FUNCTION_BLOCK FB_AnalogInput
(*
    Converts the integer from an analog input terminal to a real unit value (e.g., volts)
    2019-10-09 Zachary Lentz
*)
VAR_INPUT
    // Connect this input to the terminal
    iRaw AT %I*: INT;
    // The number of bits correlated with the terminal's max value. This is not necessarily the resolution parameter.
    iTermBits: UINT;
    // The fReal value correlated with the terminal's max value
    fTermMax: LREAL;
    // The fReal value correlated with the terminal's min value
    fTermMin: LREAL;
END_VAR
VAR_OUTPUT
    // The real value read from the output
    fReal: LREAL;
END_VAR
VAR
    fScale: LREAL;
END_VAR

IF fScale = 0 AND fTermMax > fTermMin THEN
    fScale := (EXPT(2, iTermBits) - 1) / (fTermMax - fTermMin);
END_IF
IF fScale <> 0 THEN
    fReal := iRaw / fScale + fTermMin;
END_IF

END_FUNCTION_BLOCK

(* stored: Version 1.1.0.1, ProductVersion 3.1.4022.18
   POU FB_AnalogInput: Id {c3bf2f11-e399-406d-ba95-ae8960e90a27}, SpecialFunc None *)
